{attribute 'qualified_only'}
VAR_GLOBAL
	fbParameterHandler		: Fb_ParLogging ; // Default parameter handler for visualisation and file handling
	sPARLIST_FILE			: T_MaxString 		:= 'D:\Parameters\ParameterList.csv';(* CSV destination file path and name *)
	sPARLOG_FILE			: T_MaxString 		:= 'D:\Parameters\ParameterLog.csv';(* CSV destination file path and name *)
END_VAR
VAR_GLOBAL CONSTANT
	MAX_PARAMETERS 			: UINT := 1000	;
	PAR_COLUMNS 			: UDINT := 8	;
	MAX_CSV_FIELD_LENGTH	: UDINT := 100	;
	sNetId					: T_AmsNetID		:= '' ;
END_VAR

(* stored: Version 1.1.0.1, ProductVersion 3.1.4024.11
   GVL GVL_Parameters: Id {1e32efed-448a-4ea5-a3f2-5d75543106fc} *)
